FUNCTION_BLOCK FB_System_WT_HWW_Ablaufsteuerung
VAR_IN_OUT
	Zustand					: ST_System_WT_HWW_Zustand;
	Stellwert				: ST_System_WT_HWW_Stellwert;
	Steuerung				: ST_System_WT_HWW_Steuerung;
END_VAR
VAR_INPUT
	Zustand_Regelventil_WW	: ST_RV_Zustand;
	Zustand_Stellventil_HW	: ST_SV_Zustand;
	Zustand_Pumpe_WW		: ST_PU_Zustand;
	Zustand_Pumpe_HW		: ST_PU_Zustand;
END_VAR
VAR_OUTPUT
END_VAR
VAR
	Zustand_Regelventil: BOOL;
END_VAR

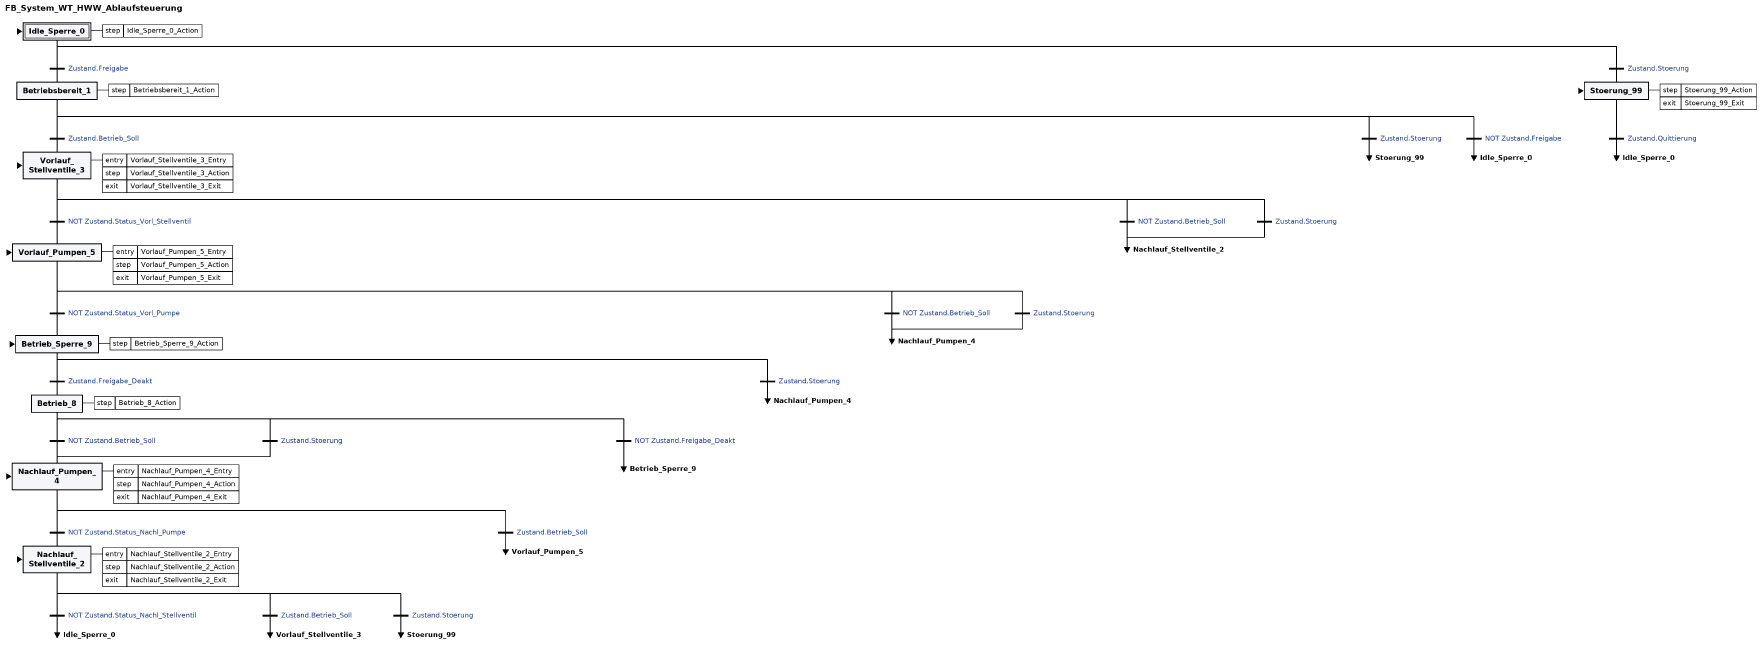
INITIAL_STEP Idle_Sperre_0:
    Idle_Sperre_0_Action(N);  // step action
END_STEP
TRANSITION FROM Idle_Sperre_0 TO Betriebsbereit_1
    := Zustand.Freigabe;
END_TRANSITION
TRANSITION FROM Idle_Sperre_0 TO Stoerung_99
    := Zustand.Stoerung;
END_TRANSITION
STEP Stoerung_99:
    Stoerung_99_Action(N);  // step action
    Stoerung_99_Exit(P0);  // exit action
END_STEP
TRANSITION FROM Stoerung_99 TO Idle_Sperre_0
    := Zustand.Quittierung;
END_TRANSITION
STEP Betriebsbereit_1:
    Betriebsbereit_1_Action(N);  // step action
END_STEP
TRANSITION FROM Betriebsbereit_1 TO Vorlauf_Stellventile_3
    := Zustand.Betrieb_Soll;
END_TRANSITION
TRANSITION FROM Betriebsbereit_1 TO Stoerung_99
    := Zustand.Stoerung;
END_TRANSITION
TRANSITION FROM Betriebsbereit_1 TO Idle_Sperre_0
    := NOT Zustand.Freigabe;
END_TRANSITION
STEP Vorlauf_Stellventile_3:
    Vorlauf_Stellventile_3_Entry(P1);  // entry action
    Vorlauf_Stellventile_3_Action(N);  // step action
    Vorlauf_Stellventile_3_Exit(P0);  // exit action
END_STEP
TRANSITION FROM Vorlauf_Stellventile_3 TO Vorlauf_Pumpen_5
    := NOT Zustand.Status_Vorl_Stellventil;
END_TRANSITION
TRANSITION FROM Vorlauf_Stellventile_3 TO Nachlauf_Stellventile_2
    := NOT Zustand.Betrieb_Soll;
END_TRANSITION
TRANSITION FROM Vorlauf_Stellventile_3 TO Nachlauf_Stellventile_2
    := Zustand.Stoerung;
END_TRANSITION
STEP Vorlauf_Pumpen_5:
    Vorlauf_Pumpen_5_Entry(P1);  // entry action
    Vorlauf_Pumpen_5_Action(N);  // step action
    Vorlauf_Pumpen_5_Exit(P0);  // exit action
END_STEP
TRANSITION FROM Vorlauf_Pumpen_5 TO Betrieb_Sperre_9
    := NOT Zustand.Status_Vorl_Pumpe;
END_TRANSITION
TRANSITION FROM Vorlauf_Pumpen_5 TO Nachlauf_Pumpen_4
    := NOT Zustand.Betrieb_Soll;
END_TRANSITION
TRANSITION FROM Vorlauf_Pumpen_5 TO Nachlauf_Pumpen_4
    := Zustand.Stoerung;
END_TRANSITION
STEP Betrieb_Sperre_9:
    Betrieb_Sperre_9_Action(N);  // step action
END_STEP
TRANSITION FROM Betrieb_Sperre_9 TO Betrieb_8
    := Zustand.Freigabe_Deakt;
END_TRANSITION
TRANSITION FROM Betrieb_Sperre_9 TO Nachlauf_Pumpen_4
    := Zustand.Stoerung;
END_TRANSITION
STEP Betrieb_8:
    Betrieb_8_Action(N);  // step action
END_STEP
TRANSITION FROM Betrieb_8 TO Nachlauf_Pumpen_4
    := NOT Zustand.Betrieb_Soll;
END_TRANSITION
TRANSITION FROM Betrieb_8 TO Nachlauf_Pumpen_4
    := Zustand.Stoerung;
END_TRANSITION
TRANSITION FROM Betrieb_8 TO Betrieb_Sperre_9
    := NOT Zustand.Freigabe_Deakt;
END_TRANSITION
STEP Nachlauf_Pumpen_4:
    Nachlauf_Pumpen_4_Entry(P1);  // entry action
    Nachlauf_Pumpen_4_Action(N);  // step action
    Nachlauf_Pumpen_4_Exit(P0);  // exit action
END_STEP
TRANSITION FROM Nachlauf_Pumpen_4 TO Nachlauf_Stellventile_2
    := NOT Zustand.Status_Nachl_Pumpe;
END_TRANSITION
TRANSITION FROM Nachlauf_Pumpen_4 TO Vorlauf_Pumpen_5
    := Zustand.Betrieb_Soll;
END_TRANSITION
STEP Nachlauf_Stellventile_2:
    Nachlauf_Stellventile_2_Entry(P1);  // entry action
    Nachlauf_Stellventile_2_Action(N);  // step action
    Nachlauf_Stellventile_2_Exit(P0);  // exit action
END_STEP
TRANSITION FROM Nachlauf_Stellventile_2 TO Idle_Sperre_0
    := NOT Zustand.Status_Nachl_Stellventil;
END_TRANSITION
TRANSITION FROM Nachlauf_Stellventile_2 TO Vorlauf_Stellventile_3
    := Zustand.Betrieb_Soll;
END_TRANSITION
TRANSITION FROM Nachlauf_Stellventile_2 TO Stoerung_99
    := Zustand.Stoerung;
END_TRANSITION

ACTION Betrieb_8_Action:
(* Stellwert setzen *)
Stellwert.Anford_Stellventil_WW	:= TRUE;
Stellwert.Anford_Stellventil_HW	:= TRUE;
Stellwert.Anford_Pumpe_WW	:= TRUE;
Stellwert.Anford_Pumpe_HW	:= TRUE;

(* Zustand setzen *)
Zustand.Status				:= E_System_WT_Zustand_Status_Betrieb;
END_ACTION

ACTION Betrieb_Sperre_9_Action:
(* Stellwert setzen *)
Stellwert.Anford_Stellventil_WW	:= TRUE;
Stellwert.Anford_Stellventil_HW	:= TRUE;
Stellwert.Anford_Pumpe_WW	:= TRUE;
Stellwert.Anford_Pumpe_HW	:= TRUE;

(* Zustand setzen *)
Zustand.Status				:= E_System_WT_Zustand_Status_Betrieb_Sperre;
END_ACTION

ACTION Betriebsbereit_1_Action:
(* Stellwert setzen *)
Stellwert.Anford_Stellventil_WW	:= FALSE;
Stellwert.Anford_Stellventil_HW	:= FALSE;
Stellwert.Anford_Pumpe_WW	:= FALSE;
Stellwert.Anford_Pumpe_HW	:= FALSE;

(* Zustand setzen *)
Zustand.Status			:= E_System_WT_Zustand_Status_Betriebsbereit;
END_ACTION

ACTION Idle_Sperre_0_Action:
(* Stellwert setzen *)
Stellwert.Anford_Stellventil_WW	:= FALSE;
Stellwert.Anford_Stellventil_HW	:= FALSE;
Stellwert.Anford_Pumpe_WW	:= FALSE;
Stellwert.Anford_Pumpe_HW	:= FALSE;

(* Zustand setzen *)
Zustand.Status			:= E_System_WT_Zustand_Status_Idle_Sperre;


(* Quittierungszustand auf False setzen, damit das System bei einer erneuten Störung nicht direkt wieder angeschaltet wird *)
Steuerung.Quittierung	:= FALSE;
END_ACTION

ACTION Nachlauf_Pumpen_4_Action:
(* Stellwert setzen *)
Stellwert.Anford_Stellventil_WW	:= TRUE;
Stellwert.Anford_Stellventil_HW	:= TRUE;
Stellwert.Anford_Pumpe_WW	:= FALSE;
Stellwert.Anford_Pumpe_HW	:= FALSE;

(* Zustand setzen *)
Zustand.Status				:= E_System_WT_Zustand_Status_Nachl_Pumpen;
Zustand.Status_Nachl_Pumpe	:= Zustand_Pumpe_WW.Betrieb OR Zustand_Pumpe_HW.Betrieb OR Zustand_Pumpe_WW.Status_Nachl OR Zustand_Pumpe_HW.Status_Nachl;
END_ACTION

ACTION Nachlauf_Pumpen_4_Entry:
Zustand.Status_Nachl_Pumpe	:= TRUE;
END_ACTION

ACTION Nachlauf_Pumpen_4_Exit:
Zustand.Status_Nachl_Pumpe	:= FALSE;
END_ACTION

ACTION Nachlauf_Stellventile_2_Action:
(* Stellwert setzen *)
Stellwert.Anford_Stellventil_WW	:= FALSE;
Stellwert.Anford_Stellventil_HW	:= FALSE;
Stellwert.Anford_Pumpe_WW	:= FALSE;
Stellwert.Anford_Pumpe_HW	:= FALSE;

(* Zustand setzen *)
Zustand.Status				:= E_System_WT_Zustand_Status_Nachl_Stellventile;
Zustand.Status_Nachl_Stellventil	:= Zustand_Stellventil_HW.Stellung OR Zustand_Stellventil_HW.Stellungwechsel10;
END_ACTION

ACTION Nachlauf_Stellventile_2_Entry:
Zustand.Status_Nachl_Stellventil	:= TRUE;
END_ACTION

ACTION Nachlauf_Stellventile_2_Exit:
Zustand.Status_Nachl_Stellventil	:= FALSE;
END_ACTION

ACTION Stoerung_99_Action:
(* Stellwert setzen *)
Stellwert.Anford_Stellventil_WW	:= FALSE;
Stellwert.Anford_Stellventil_HW	:= FALSE;
Stellwert.Anford_Pumpe_WW	:= FALSE;
Stellwert.Anford_Pumpe_HW	:= FALSE;

(* Zustand setzen *)
Zustand.Stoerung			:= TRUE;
Zustand.Status			:= E_System_WT_Zustand_Status_Stoerung;
END_ACTION

ACTION Stoerung_99_Exit:
Zustand.Stoerung	:= FALSE;
END_ACTION

ACTION Vorlauf_Pumpen_5_Action:
(* Stellwert setzen *)
Stellwert.Anford_Stellventil_WW	:= TRUE;
Stellwert.Anford_Stellventil_HW	:= TRUE;
Stellwert.Anford_Pumpe_WW	:= TRUE;
Stellwert.Anford_Pumpe_HW	:= TRUE;

(* Zustand setzen *)
Zustand.Status				:= E_System_WT_Zustand_Status_Vorl_Pumpen;
Zustand.Status_Vorl_Pumpe	:= NOT(Zustand_Pumpe_WW.Betrieb AND Zustand_Pumpe_HW.Betrieb AND NOT Zustand_Pumpe_WW.Status_Vorl AND NOT Zustand_Pumpe_HW.Status_Vorl);
END_ACTION

ACTION Vorlauf_Pumpen_5_Entry:
Zustand.Status_Vorl_Pumpe	:= TRUE;
END_ACTION

ACTION Vorlauf_Pumpen_5_Exit:
Zustand.Status_Vorl_Pumpe	:= FALSE;
END_ACTION

ACTION Vorlauf_Stellventile_3_Action:
(* Stellwert setzen *)
Stellwert.Anford_Stellventil_WW	:= TRUE;
Stellwert.Anford_Stellventil_HW	:= TRUE;
Stellwert.Anford_Pumpe_WW	:= FALSE;
Stellwert.Anford_Pumpe_HW	:= FALSE;

(* Zustand setzen *)
Zustand.Status				:= E_System_WT_Zustand_Status_Vorl_Stellventile;
Zustand.Status_Vorl_Stellventil	:= NOT(Zustand_Stellventil_HW.Stellung AND NOT Zustand_Stellventil_HW.Stellungwechsel01);
END_ACTION

ACTION Vorlauf_Stellventile_3_Entry:
Zustand.Status_Vorl_Stellventil	:= TRUE;
END_ACTION

ACTION Vorlauf_Stellventile_3_Exit:
Zustand.Status_Vorl_Stellventil	:= FALSE;
END_ACTION

END_FUNCTION_BLOCK

(* stored: Version 1.1.0.1, ProductVersion 3.1.4024.9
   POU FB_System_WT_HWW_Ablaufsteuerung: Id {541511f7-c164-4e14-a889-acc4aef4abbb}, SpecialFunc None
   Action Betrieb_8_Action: Id {c3af29be-8557-44e8-97f0-c01edaed8956}
   Action Betrieb_Sperre_9_Action: Id {d1db82f0-0543-420e-9413-5a10c777b3d9}
   Action Betriebsbereit_1_Action: Id {d7997101-5e2e-45c4-ac32-5951a978aa01}
   Action Idle_Sperre_0_Action: Id {7374cb44-8eb5-4946-8ec1-fb016b8d1a69}
   Action Nachlauf_Pumpen_4_Action: Id {41306168-6c55-49ed-aab6-50afa1e321a8}
   Action Nachlauf_Pumpen_4_Entry: Id {d9e28a78-4d66-4140-bdc4-3c7f62400ec1}
   Action Nachlauf_Pumpen_4_Exit: Id {e661972a-0757-4fef-b7ab-f6bc3b8777df}
   Action Nachlauf_Stellventile_2_Action: Id {5f3d107e-5746-45ae-affa-457f4f63386e}
   Action Nachlauf_Stellventile_2_Entry: Id {5cb2ec00-b2a0-4509-aef3-ea67f51ac27b}
   Action Nachlauf_Stellventile_2_Exit: Id {454e7e51-4c4b-4886-b673-7117301d5996}
   Action Stoerung_99_Action: Id {8156ffa6-02e8-4e21-ad05-5dacc1310367}
   Action Stoerung_99_Exit: Id {2cf1fb09-88cf-4865-8e32-5548b5c4c286}
   Action Vorlauf_Pumpen_5_Action: Id {fab8a4a2-64c7-4379-b152-45d1c6af23e2}
   Action Vorlauf_Pumpen_5_Entry: Id {d80c2979-d8f0-4a2c-8a05-b53e3f95b761}
   Action Vorlauf_Pumpen_5_Exit: Id {024fd589-bf82-49e2-87cc-a737f620d4dc}
   Action Vorlauf_Stellventile_3_Action: Id {99fd4986-ed17-4996-b565-5da9f0e11038}
   Action Vorlauf_Stellventile_3_Entry: Id {a606a1f1-c9ae-44ab-aa07-064cd7c14b77}
   Action Vorlauf_Stellventile_3_Exit: Id {416b20b6-34d8-4703-bd25-872fd9d430d3} *)
